(* IEC 61131-3 sources: ICSQuartz/benchmarks/oscat_basic_weekday_to_string/src, 1 file *)

(* ---- program.st ---- *)
PROGRAM PLC_PRG
VAR_INPUT
    in_WDAY: INT;
    in_LANG: INT;
    in_LX: INT;
END_VAR

WEEKDAY_TO_STRING(in_WDAY, in_LANG, in_LX);

END_PROGRAM
